// TwinCAT 3 PLC project testStepper
// ProgramVersion: 3.1.4023.0
// libraries:
//   Tc2_MC2, * (Beckhoff Automation GmbH)
//   Tc2_NC, * (Beckhoff Automation GmbH)
//   Tc2_Standard, * (Beckhoff Automation GmbH)
//   Tc2_System, * (Beckhoff Automation GmbH)
//   Tc3_Module, * (Beckhoff Automation GmbH)
//   VisuDialogs, * (System)
// project tree:
//   GlobalPOUs/ MAIN.TcPOU (not stored)
//   / GlobalTextList.TcGTLO, PlcTask.TcTTO, Visualization Manager.TcVMO (not stored)
//   GVLs/ GVL_AxisCtr.TcGVL (not stored), GVL_IO.TcGVL (not stored), GVL_NC.TcGVL
//   Motion_POUs/ Command_to_Action.TcPOU (not stored), DegreesToRelativeMovment.TcPOU (not stored), movements.TcPOU (not stored), PositionToDegree.TcPOU (not stored), POUNCPowerOn.TcPOU (not stored), Torque_reading.TcPOU
//   VISUs/ testStepperVisu.TcVIS (not stored)
// real-time tasks:
//   TASK PlcTask: cycle T#10ms, priority 21, ADS port 350
// motion (NC):
//   TASK NC-SteeringAxis SAF: cycle T#2ms, priority 4, ADS port 501
//   TASK NC-SteeringAxis SVB: cycle T#10ms, priority 8, ADS port 511
//   AXIS Axis 1 (id 1)
//     OtherSettings: AllowMotionCmdToSlave=true
//     encoder EncType=1
//     drive DrvType=5
//       Analog: TorqueSetpointScale=10, ScaleFactorActTorque=0.1
//       TimeComp: TaskDelayCycles=1
//     controller CtrType=1
//       CtrPara: PriorControlFactor=1
//         Observer: BandWidth=20

CONFIGURATION testStepper
    RESOURCE PLC ON TwinCAT3
        TASK PlcTask(INTERVAL := T#10ms, PRIORITY := 21);
        PROGRAM MAIN WITH PlcTask : MAIN;
    END_RESOURCE
END_CONFIGURATION

// ---- GVLs/GVL_NC.TcGVL
{attribute 'qualified_only'}
VAR_GLOBAL
	stXAxis :AXIS_REF;
	stXaxisStatus : ST_AxisStatus;
	
END_VAR

// ---- Motion_POUs/Torque_reading.TcPOU
PROGRAM Torque_reading
VAR
	MC_TorqueControl_0: MC_TorqueControl;
END_VAR

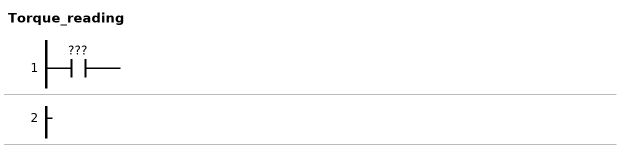
// NETWORK 1

// NETWORK 2

END_PROGRAM

// ---- GlobalTextList.TcGTLO
TEXTLIST GlobalTextList
  163 = '%10.1f'
  781 = '%1f'
  35 = '%d'
  559 = '%d s'
  953 = '%i'
  523 = 'EndSwitch'
  895 = 'Execute'
  52 = 'Reset'
  627 = 'setAngle'
  485 = 'Start Homing'
  860 = 'StartHoming'
  447 = 'X-Axis enable'
  34 = 'x-axis limit+'
  942 = 'x-axis limit-'
END_TEXTLIST
